INTERFACE I_Asset

METHOD add_template_job : BOOL
VAR_INPUT
	template_job : I_JobCatalogue;
END_VAR
END_METHOD

PROPERTY asset_kind : E_AssetKind
GET
END_GET
SET
END_SET
END_PROPERTY

PROPERTY asset_name : STRING
GET
END_GET
SET
END_SET
END_PROPERTY

METHOD asset_start : BOOL
VAR_INPUT
END_VAR
END_METHOD

PROPERTY driver : I_Job
SET
END_SET
END_PROPERTY

PROPERTY error_id : HRESULT
GET
END_GET
END_PROPERTY

PROPERTY iter_process_jobs : I_JobCatalogue
GET
END_GET
END_PROPERTY

METHOD process_job_start : BOOL
VAR_INPUT
END_VAR
END_METHOD

METHOD remove_template_job_by_name : BOOL
VAR_INPUT
	template_name : T_MaxString;
END_VAR
END_METHOD

METHOD remove_template_job_by_object : BOOL
VAR_INPUT
	template_job : I_JobCatalogue;
END_VAR
END_METHOD

METHOD select_process_job : BOOL;
VAR_INPUT
	template_name : T_MaxString;
END_VAR
END_METHOD

PROPERTY selected_process_job : I_Job
GET
END_GET
END_PROPERTY

METHOD set_parameters : BOOL
VAR_INPUT
END_VAR
END_METHOD

END_INTERFACE

(* stored: Version 1.1.0.1, ProductVersion 3.1.4026.13
   Itf I_Asset: Id {12ee3a8b-6456-41e5-84b8-0def38f5c9f0}
   Method add_template_job: Id {37e01327-d2bd-46ce-b321-590953217d5a}
   Property asset_kind: Id {10644835-1f1e-45a8-a601-a3d47cf7ad6c}
   Get Get: Id {b28c6d47-d324-4fb8-93b4-dc0bbc1dad9d}
   Set Set: Id {89cc2090-3bb8-4d8e-bf55-1a53e65ee35c}
   Property asset_name: Id {e2cdb12b-c064-464e-9d9a-1116554bf7b9}
   Get Get: Id {b696988b-4321-4ae1-ae35-024b551a560a}
   Set Set: Id {9685391f-b9a8-4bf9-946f-a226839fa52d}
   Method asset_start: Id {aefe3fdb-0823-4b31-acac-ea1574422993}
   Property driver: Id {5e18b4e8-e6c4-4f9e-8aad-5a99d742e6ab}
   Set Set: Id {5e1ddfc0-20b4-46da-a731-9c6837509368}
   Property error_id: Id {f8c642f5-2f6c-4dc4-8d68-871d75d4fbe2}
   Get Get: Id {981e5c57-44b0-44b5-90b2-f01952fffb78}
   Property iter_process_jobs: Id {7109d664-7ce1-4fe0-886e-bf8e706f61a3}
   Get Get: Id {e6044fb6-ed53-4327-85dc-8f6ad671ea19}
   Method process_job_start: Id {684b9a85-e17f-4e1e-9a23-ae4a88fa35be}
   Method remove_template_job_by_name: Id {17291b40-2ac9-483d-8762-5d3ace7184cb}
   Method remove_template_job_by_object: Id {222e0364-4f8a-40ec-babf-c76b4a6f5ce0}
   Method select_process_job: Id {dc80ce92-6ddb-4acd-b37b-3f2900d56045}
   Property selected_process_job: Id {a3431bac-dd92-47ec-8489-56c0f1e36cde}
   Get Get: Id {1b07124f-bdef-4872-8368-148cea1db887}
   Method set_parameters: Id {fc43c4b4-f32f-496c-9367-1e89e763c2d2} *)
